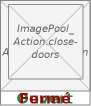
VISUALIZATION Door  // 91x106
VAR_IN_OUT
	Etat_MaAr	:BOOL;
END_VAR
    Rectangle (15,91 60x15), "Ouvert", invisible if: Etat_MaAr, text list: 'OuvFerm', text index: S_Cmd_ElectroValve_Alim_Lavabo
    Rectangle (15,91 60x15), "Fermé", invisible if: NOT Etat_MaAr, text list: 'OuvFerm', text index: S_Cmd_ElectroValve_Alim_Lavabo
    Image (0,0 91x91), invisible if: Etat_MaAr, image: ImagePool_Action.door-open
    Image (8,4 75x75), invisible if: NOT Etat_MaAr, image: ImagePool_Action.close-doors
END_VISUALIZATION

(* stored: Version 1.1.0.1, ProductVersion 3.1.4024.15
   Visu Door: Id {3d3f7174-d3f3-4094-9738-3ecb8fe11067} *)
